PROGRAM MAIN
VAR
	pTemperature : fbRaiseTemperature;
END_VAR


dbIO.bWriteEnable:=TRUE;

pTemperature(bReset := dbIO.bReset,
			bAlarm => dbIO.bAlarm,
			rTemperature => dbIO.rTemperature);

END_PROGRAM

(* stored: Version 1.1.0.1, ProductVersion 3.1.4024.12
   POU MAIN: Id {15c42c1c-5789-41aa-83cc-1ff2f55013d4}, SpecialFunc None *)
